// ---- POUs/FB_WaterFill.TcPOU
//=============================================================================
// FB_WaterFill | VERIFIED 7.30.26 DA
//-----------------------------------------------------------------------------
//
// TWO modes selected by eMode:
//
//   StartupFill
//     - Open SV4 while the filtered CENTER switch (LS1) is dry.
//     - The instant LS1 is covered, CLOSE SV4 and run a fixed confirm dwell
//       (legacy T24 = 5 s). Valve does NOT keep filling during the dwell.
//     - When the dwell completes -> bFillComplete.
//     - If the fill-fault timer (legacy T10, preset tFillFaultTime) expires
//       while LS1 is still dry -> bWaterFillFault (legacy B1600.15 -> S10).
//
//   RunningAutofill
//     - A self-contained PID holds level at the center switch (setpoint 25).
//       Its output % is time-proportioned onto the on/off solenoid over
//       tFillCycle (legacy T20 / V1516) -> metered trickle to replace boil-off.
//     - Lower-duty floor: below rFillMinDuty (legacy 10%) the valve
//       stays shut - no meaningless sub-threshold pulsing.
//     - If the PID sits pinned at full output longer than tWaterFillCheck -> bWaterRegFault
//
// Switch filtering: raw center/empty switches debounced with
// symmetric on/off delays (tLevelFilter).
//
// Drives NO coil directly. Outputs qFillValve; FB_OutputHandler (single
// writer) maps it to GVL_IO
//
//=============================================================================
FUNCTION_BLOCK FB_WaterFill
VAR_INPUT
    eMode            : E_WaterFillMode;   // StartupFill | RunningAutofill | Idle
	rSteamFlow		 : REAL;
    bCenterSwitch    : BOOL;              // RAW LS1 center (X2). Filtered internally.
    bEmptySwitch     : BOOL;              // RAW LS3 empty  (X4). Filtered internally.
    bAutofillEnable  : BOOL;              // legacy X13 autofill-off signal
END_VAR
VAR_OUTPUT
    qFillValve       : BOOL;              // -> FB_OutputHandler -> SV4
    bFillComplete    : BOOL;              // startup fill done (LS1 covered + dwell)
    bCenterFiltered  : BOOL;              // exposed filtered LS1 (HMI / diagnostics)
    bEmptyFiltered   : BOOL;              // exposed filtered LS3
END_VAR
VAR
    // ---- switch debounce (symmetric on/off = tLevelFilter) ----
    tonCenterOn      : TON;
    tonCenterOff     : TON;
    tonEmptyOn       : TON;
    tonEmptyOff      : TON;
	
	// autofill switch delay timers
	tonCenterOn_Autofill : TON;
	tonCenterOff_Autofill : TON;

    // ---- startup fill (K8) -------------------------------------------------
    tonFillDwell     : TON; // fixed confirm (tFillConfirm = 5 s)

    // ---- running autofill (K7) ---------------------------------------------
    tonAutoFillDwell : TON;	// legacy T63, preset tWaterFillCheck (V1555)
	bAutoFillActive	 : BOOL;

    ePrevMode        : E_WaterFillMode;
    bModeEntry       : BOOL;
	
	rWaterLevel		 : REAL;
	rOutputPct		 : REAL;
	rDrainFactor	 : REAL := 0.1;
	rFillFactor	 	 : REAL := 1;
	
	// --- PID sample-rate gate -----------------------------------------------
    fbSampleTick        : TON;
    bSample             : BOOL;
    rDt                 : REAL;              // [s] sample interval as a real
	
    // --- per-loop PID state (index = legacy PID number) --------------------
    rIntegral          : REAL;
    rPrevPv            : REAL;
    rPrimed            : BOOL;

    // --- per-loop PWM state -------------------------------------------------
    tonPwmTimer          :  TON;
    rPwmDutyLatched    :  REAL;

    i                   : INT;
	
END_VAR

// mode-entry edge: reset per-mode timers/faults when the mode changes so a
// second entry never sees stale .Q or accumulated time.
bModeEntry := (eMode <> ePrevMode);
ePrevMode  := eMode;

//============================================================================
// 1. SWITCH DEBOUNCE  (symmetric on/off delay = tLevelFilter)
//============================================================================
tonCenterOn (IN := bCenterSwitch,     PT := GVL_SysParameters.tDebounceTimer);
tonCenterOff(IN := NOT bCenterSwitch, PT := GVL_SysParameters.tDebounceTimer);
IF tonCenterOn.Q THEN
    bCenterFiltered := TRUE;
ELSIF tonCenterOff.Q THEN
    bCenterFiltered := FALSE;
END_IF

tonEmptyOn (IN := bEmptySwitch,     PT := GVL_SysParameters.tDebounceTimer);
tonEmptyOff(IN := NOT bEmptySwitch, PT := GVL_SysParameters.tDebounceTimer);
IF tonEmptyOn.Q THEN
    bEmptyFiltered := TRUE;
ELSIF tonEmptyOff.Q THEN
    bEmptyFiltered := FALSE;
END_IF

//============================================================================
// 2. MODE LOGIC
//============================================================================
CASE eMode OF

    //-- STARTUP FILL ------------------------------------------
    E_WaterFillMode.StartupFill:
        IF bModeEntry THEN
            bFillComplete   := FALSE;
            tonFillDwell(IN := FALSE);
        END_IF

        IF NOT bCenterFiltered THEN
            // --- still filling: valve open, fault timer running ---
            qFillValve := TRUE;
        ELSE
            // --- LS1 covered: CLOSE valve immediately, run confirm dwell ---
            // (legacy rung 502: RST Y4 on the same rung TMR T24 starts)
            tonFillDwell(IN := bCenterFiltered, PT := GVL_SysParameters.tStartupFillDelay);
			IF tonFillDwell.Q THEN
				qFillValve := FALSE;
				bFillComplete := TRUE;
			END_IF
        END_IF

    //-- RUNNING AUTOFILL --------------------------------------
    E_WaterFillMode.RunningAutofill:
        IF bModeEntry THEN
			tonAutoFillDwell(IN := FALSE);
        END_IF

        (*IF NOT bAutofillEnable THEN
            // autofill off -> valve closed, timers reset
            qFillValve := FALSE;    
		ELSE
			IF NOT bCenterFiltered THEN
				qFillValve := TRUE;
				tonAutoFillDwell(IN := FALSE);
			ELSE
				tonAutoFillDwell(IN := TRUE, PT := GVL_SysParameters.tAutoFillDelay);
				IF tonAutoFillDwell.Q THEN
					qFillValve := FALSE;
				END_IF
			END_IF
        END_IF *)
//----------------------------//

		
		fbSampleTick(IN := NOT fbSampleTick.Q, PT := GVL_SysParameters.tAutofillPidSample);
		bSample := fbSampleTick.Q;
		rDt     := UDINT_TO_REAL(TIME_TO_UDINT(GVL_SysParameters.tPidSampleTime)) * 0.001;
				
	
		IF NOT bAutofillEnable THEN
			qFillValve := FALSE;
		ELSE
			tonCenterOn_Autofill(IN := bCenterSwitch, PT := T#2M);
			tonCenterOff_Autofill(IN := NOT bCenterSwitch, PT := T#2M);
			
			
			IF bSample THEN
				rOutputPct := RunPid(
										 rSp       := 25,
										 rPv       := rWaterLevel,
										 rKp       := 5.0,
										 rTi       := GVL_SysParameters.rPid1_Ti,
										 rTd       := GVL_SysParameters.rPid1_Td,
										 rOutMin   := 5.0,
										 rOutMax   := 35.0,
										 rDt       := rDt);
										 
				rWaterLevel := rWaterLevel - rSteamFlow * rDrainFactor + rOutputPct * rFillFactor;
				rWaterLevel := LIMIT(0.0, rWaterLevel, 100.0);
			END_IF
			
			IF tonCenterOn_Autofill.Q THEN rOutputPct := 0; END_IF
			IF tonCenterOff_Autofill.Q THEN rOutputPct := 35; END_IF
			qFillValve := RunPwm(rDutyPct := rOutputPct);
				 
	
		END_IF

    //-- IDLE --------------------------------------------------------------
    ELSE
        qFillValve := FALSE;
        tonFillDwell(IN := FALSE);
END_CASE

//=============================================================================
// RunPid
//-----------------------------------------------------------------------------
// Standard (ISA) positional PID, output in percent.
//
//   out = Kp * e  +  (Kp/Ti) * INTEGRAL(e)  -  Kp * Td * d(PV)/dt
//
// Derivative acts on the MEASUREMENT, not the error, so a setpoint change
// does not produce a derivative spike.
//
// Anti-windup: the integral accumulator is clamped to the output range. This
// is the same trick as legacy rung 456 ("freeze integral if over"), which
// clamped the PID bias word to the output maximum.
//
// State lives in the FB's arrays, indexed by nLoop, so one method serves
// every loop. Call at the sample rate only - it uses rDt, not the task cycle.
//=============================================================================
METHOD PRIVATE RunPid : REAL
VAR_INPUT
    rSp     : REAL;     // setpoint, engineering units
    rPv     : REAL;     // process value, same units
    rKp     : REAL;     // proportional gain [% per engineering unit]
    rTi     : REAL;     // integral / reset time [s]. 0 disables integral action
    rTd     : REAL;     // derivative / rate time [s]. 0 disables derivative
    rOutMin : REAL;     // output floor [%]
    rOutMax : REAL;     // output ceiling [%]
    rDt     : REAL;     // sample interval [s]
END_VAR
VAR_INST
    rError  : REAL;
    rProp   : REAL;
    rDeriv  : REAL;
    rOut    : REAL;
END_VAR
rError := rSp - rPv;

//--- proportional ------------------------------------------------------------
rProp := rKp * rError;

//--- integral ----------------------------------------------------------------
IF rTi > 0.0 THEN
    rIntegral := rIntegral + (rKp / rTi) * rError * rDt;
    // clamp to the output range: prevents wind-up while saturated
    rIntegral := LIMIT(rOutMin, rIntegral, rOutMax);
ELSE
    rIntegral := 0.0;
END_IF

//--- derivative on measurement ------------------------------------------------
// Skipped on the first sample after a reset, when arPrevPv is meaningless.
IF (rTd > 0.0) AND rPrimed THEN
    rDeriv := -rKp * rTd * (rPv - rPrevPv) / rDt;
ELSE
    rDeriv := 0.0;
END_IF
rPrevPv := rPv;
rPrimed := TRUE;

//--- sum and clamp ------------------------------------------------------------
rOut   := rProp + rIntegral + rDeriv;
RunPid := LIMIT(rOutMin, rOut, rOutMax);
END_METHOD

//=============================================================================
// RunPwm
//-----------------------------------------------------------------------------
// Time-proportioned output: turns a 0..100 % demand into a digital heater
// command with a fixed period. 
//
// The demand is LATCHED at each period boundary. Without this the
// on-time would move underneath an in-progress pulse.
//
// Must be called EVERY task cycle - the period timer only advances when it
// is called. Resolution is one task cycle (10 ms), so a 2 s period gives
// 0.5 % granularity.
//=============================================================================
METHOD PRIVATE RunPwm : BOOL
VAR_INPUT
    rDutyPct : REAL;    // demand 0..100 %
    
END_VAR
VAR_INST
	tPeriod   : TIME := T#2S;    
    nPeriodMs : UDINT;
    nOnMs     : UDINT;
    rDuty     : REAL;
END_VAR
nPeriodMs := TIME_TO_UDINT(tPeriod);

//--- free-running period timer -----------------------------------------------
// IN := NOT Q self-restarts the TON: Q is true for one cycle, which drops IN,
// which clears ET. Costs one task cycle per period (0.5 % at 2 s).
tonPwmTimer(IN := NOT tonPwmTimer.Q, PT := tPeriod);

//--- latch the demand once per period ----------------------------------------
// ET is only zero at a period boundary (and on the very first call), so this
// refreshes the on-time exactly once per pulse and never mid-pulse.
IF tonPwmTimer.ET = T#0S THEN
    rDuty := rDutyPct;
END_IF

rDuty := LIMIT(0.0, rDuty, 100.0);

//--- resolve the pulse --------------------------------------------------------
IF rDuty <= 0.0 THEN
    RunPwm := FALSE;
ELSIF rDuty >= 100.0 THEN
    // Special-cased so a saturated loop holds the coil solid instead of
    // dropping out for the single cycle it takes the timer to roll over.
    RunPwm := TRUE;
ELSE
    nOnMs  := REAL_TO_UDINT(rDuty * 0.01 * UDINT_TO_REAL(nPeriodMs));
    RunPwm := TIME_TO_UDINT(tonPwmTimer.ET) < nOnMs;
END_IF
END_METHOD

END_FUNCTION_BLOCK

// ---- POUs/FB_OutputHandler.TcPOU
FUNCTION_BLOCK FB_OutputHandler
VAR_INPUT
    eState           : E_SystemState;

    // --- automatic sources (intent from control/sequence FBs) ---
    bWaterFillValve	 : BOOL;	// FB_WaterFill request  -> SV4
    bPurgeValve      : BOOL;	// FB_Purge request      -> SV2 during purge
    bDeliveryPermit  : BOOL;	// state machine: SV3 delivery allowed
    bH1Upstream      : BOOL;	// upstream heater
    bH2Purifier      : BOOL;	// spa haeter
    bFmHeater        : BOOL;	// flowmeter heater
    bExtHeater       : BOOL;	// external heater

    // --- maintenance overrides (FALSE outside Maintenance; gated in FB_Hmi) ---
    arValveOverride  : ARRAY[1..4] OF BOOL;   // 1=SV1 2=SV2 3=SV3 4=SV4

    // --- process feedback needed for actuation timing ---
    stProcess        : ST_ProcessValues;
END_VAR
VAR_OUTPUT
    // feedback for HMI (what we actually commanded this cycle)
    arValveState     : ARRAY[1..4] OF BOOL;
    bHeatersOn       : BOOL;
END_VAR
VAR
    // resolved valve commands before interlocks
    bSV1_DrainValve        	: BOOL;
    bSV2_SpaValve          	: BOOL;
    bSV3_DeliveryValve     	: BOOL;
    bSV4_WaterInletValve   	: BOOL;

    // SesOff SV2 pressure relief delayed close
    tonSv2Close      		: TON;

    bRunningState    		: BOOL;
END_VAR

// Convenience: are we in a state that runs process automatically?
bRunningState := (eState = E_SystemState.FillWater)
              OR (eState = E_SystemState.PurgeVessel)
              OR (eState = E_SystemState.SetDiffPressure)
              OR (eState = E_SystemState.InitMain)
              OR (eState = E_SystemState.SteamFlowing);

//============================================================================
// 1. RESOLVE VALVE COMMANDS BY CONTEXT  (all boolean - solenoids are on/off)
//============================================================================
CASE eState OF

    //-- Manual mode: HMI overrides drive the valves directly --------------
    E_SystemState.Maintenance:
        bSV1_DrainValve    		:= arValveOverride[1];
        bSV2_SpaValve      		:= arValveOverride[2];
        bSV3_DeliveryValve 		:= arValveOverride[3];
        bSV4_WaterInletValve    := arValveOverride[4];

    //-- Safe shutdown: SV1/3/4 closed; SV2 pressure-relief then delayed ----
    //   SV2 held open until upstream pressure < 800 Torr
    E_SystemState.SesOff, E_SystemState.InitController, E_SystemState.CheckIfHot, E_SystemState.Fault:
        bSV1_DrainValve    := FALSE;
        bSV3_DeliveryValve := FALSE;
        bSV4_WaterInletValve    := FALSE;
        tonSv2Close(IN := (stProcess.rPt1Upstream < GVL_SysParameters.rUpstreamPressureReleived),
                    PT := GVL_SysParameters.tSv2CloseDelay);
        bSV2_SpaValve := NOT tonSv2Close.Q;   // stay open until relieved+delay

    //-- Running states: automatic intent from sequence FBs ------------------
    ELSE
        tonSv2Close(IN := FALSE);   // keep the relief timer reset while running
		
		// SV1 drain: closed in these states (drain handled via maintenance)
        bSV1_DrainValve := bPurgeValve;

        // SV2 main: open during purge, and held open while steam is flowing
        bSV2_SpaValve := TRUE;

        // SV3 process delivery: pure on/off. Legacy Y3 is SET on SES-On and
        // RST on SES-Off / stage exit. Here the state machine supplies the
        // delivery permit; SV3 opens only while flowing and permitted.
        bSV3_DeliveryValve := (eState = E_SystemState.SteamFlowing) AND bDeliveryPermit;

        // Water fill sequence owns SV4
        bSV4_WaterInletValve := bWaterFillValve;

END_CASE

//============================================================================
// 2. HARD INTERLOCKS  (apply AFTER resolution; no state can bypass)
//============================================================================
IF bSV3_DeliveryValve THEN
    bSV1_DrainValve := FALSE;         // no draining during delivery
END_IF
IF bSV1_DrainValve THEN
    bSV2_SpaValve := FALSE;          // isolate main while draining
END_IF

//============================================================================
// 3. RESOLVE HEATERS
//============================================================================
// Heaters run ONLY in running states. In SesOff/Fault/Maint heaters are off
IF NOT bRunningState THEN
    bH1Upstream := FALSE;
    bH2Purifier := FALSE;
    bFmHeater   := FALSE;
    bExtHeater  := FALSE;
END_IF

//============================================================================
// 4. SINGLE WRITE POINT -> physical coils
//============================================================================
GVL_IO.boSV1_DrainValve         := bSV1_DrainValve;
GVL_IO.boSV2_SpaValve           := bSV2_SpaValve;
GVL_IO.boSV3_DeliveryValve      := bSV3_DeliveryValve;
GVL_IO.boSV4_WaterInletValve	:= bSV4_WaterInletValve;

GVL_IO.boH1_UpstreamHeater 		:= bH1Upstream;
GVL_IO.boH2_SpaHeater 			:= bH2Purifier;
GVL_IO.boH3_FlowmeterHeater 	:= bFmHeater;
GVL_IO.boH4_ExternalHeater		:= bExtHeater;

//============================================================================
// 5. FEEDBACK for HMI
//============================================================================
arValveState[1] := bSV1_DrainValve;
arValveState[2] := bSV2_SpaValve;
arValveState[3] := bSV3_DeliveryValve;
arValveState[4] := bSV4_WaterInletValve;
bHeatersOn := bH1Upstream OR bH2Purifier OR bFmHeater OR bExtHeater;

END_FUNCTION_BLOCK
